TYPE T_Query_Interface : __SYSTEM.IQueryInterface; END_TYPE

(* stored: Version 1.1.0.1, ProductVersion 3.1.4022.18
   DUT T_Query_Interface: Id {612088b5-abe5-4008-a87b-38d41d5ce749} *)
